{attribute 'qualified_only'}
{attribute 'strict'}
TYPE FeedingState :
(
	State_Init 					,
	State_AutoStart         	,
	State_AutoHysterisis    	,
	State_AutoStop          	,
	State_AutoTopSensorReached 	,
	State_AutoFinalPosition     ,
	State_AutoBackToInit        ,
	State_Feeding				,
	State_Override				,
	State_Error					,
	State_ManualMoveUp			,
	State_ManualMoveDown    	
 
);
END_TYPE

(* stored: Version 1.1.0.1, ProductVersion 3.1.4024.12
   DUT FeedingState: Id {c893dbe9-bafd-4cd0-9c79-c8c4b2aead78} *)
